# EPICS autosave request: RigakuApp/Db/ADRigaku_settings.req
$(P)$(R)FlatFieldCorrection
$(P)$(R)Redistribution
$(P)$(R)OuterEdge
$(P)$(R)Pileup
$(P)$(R)PixelCorrection
$(P)$(R)CountingRate
$(P)$(R)InterChip
$(P)$(R)ImageMode
$(P)$(R)TriggerMode
$(P)$(R)UpperThreshold
$(P)$(R)LowerThreshold
$(P)$(R)AcquisitionDelay
$(P)$(R)ExposureDelay
$(P)$(R)ExposureInterval
$(P)$(R)CalibrationLabel
$(P)$(R)Username
$(P)$(R)Password
$(P)$(R)FilePath
$(P)$(R)FileName
$(P)$(R)Corrections

file "ADBase_settings.req", "P=$(P), R=$(R)
